// TIA Portal V20 export
ORGANIZATION_BLOCK "Main"   // OB124, LAD, ProgramCycle
TITLE = "Main Program Sweep (Cycle)"
// stored: Namespace PFE, SetENOAutomatically false
   VAR_INPUT
      Initial_Call : Bool;   // Initial call of this OB
      Remanence : Bool;   // =True, if remanent data are available
   END_VAR
   VAR_TEMP
      tempEnable : Bool;   // Replace with the user tags
      tempFilter : Bool;   // Replace with the user tags
      tempValid : Bool;   // Replace with the user tags
      tempBusy : Bool;   // Replace with the user tags
      tempError : Bool;   // Replace with the user tags
      tempStatus : Word;   // Replace with the user tags
   END_VAR
BEGIN

REGION Network 1: Calling Digital Event Handler
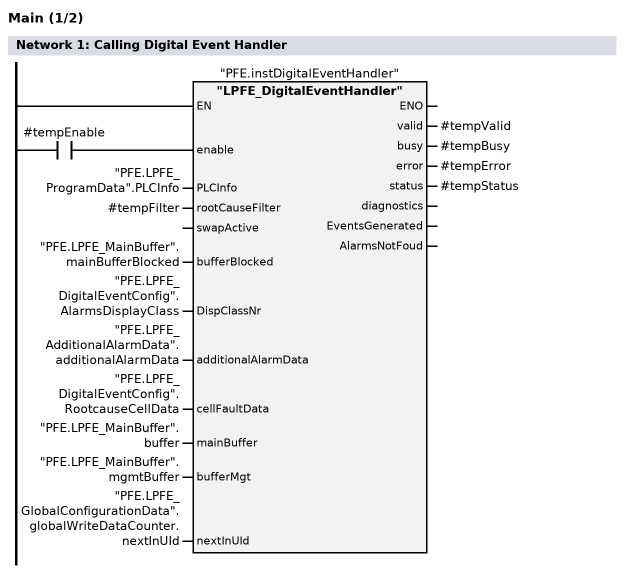
   RUNG wire#powerrail
      "PFE.instDigitalEventHandler"(enable := wire#w1, PLCInfo := "PFE.LPFE_ProgramData".PLCInfo, rootCauseFilter := #tempFilter, swapActive :=, bufferBlocked := "PFE.LPFE_MainBuffer".mainBufferBlocked, DispClassNr := "PFE.LPFE_DigitalEventConfig".AlarmsDisplayClass, additionalAlarmData := "PFE.LPFE_AdditionalAlarmData".additionalAlarmData, cellFaultData := "PFE.LPFE_DigitalEventConfig".RootcauseCellData, mainBuffer := "PFE.LPFE_MainBuffer".buffer, bufferMgt := "PFE.LPFE_MainBuffer".mgmtBuffer, nextInUId := "PFE.LPFE_GlobalConfigurationData".globalWriteDataCounter.nextInUId, valid => #tempValid, busy => #tempBusy, error => #tempError, status => #tempStatus, diagnostics =>, EventsGenerated =>, AlarmsNotFoud =>)
   END_RUNG
   RUNG wire#powerrail
      Contact( #tempEnable )
   END_RUNG wire#w1
   // the same network as SCL:
   "PFE.instDigitalEventHandler"(enable := #tempEnable,   // "LPFE_DigitalEventHandler"
                           PLCInfo := "PFE.LPFE_ProgramData".PLCInfo,
                           rootCauseFilter := #tempFilter,
                           bufferBlocked := "PFE.LPFE_MainBuffer".mainBufferBlocked,
                           DispClassNr := "PFE.LPFE_DigitalEventConfig".AlarmsDisplayClass,
                           additionalAlarmData := "PFE.LPFE_AdditionalAlarmData".additionalAlarmData,
                           cellFaultData := "PFE.LPFE_DigitalEventConfig".RootcauseCellData,
                           mainBuffer := "PFE.LPFE_MainBuffer".buffer,
                           bufferMgt := "PFE.LPFE_MainBuffer".mgmtBuffer,
                           nextInUId := "PFE.LPFE_GlobalConfigurationData".globalWriteDataCounter.nextInUId,
                           valid => #tempValid,
                           busy => #tempBusy,
                           error => #tempError,
                           status => #tempStatus);
END_REGION

REGION Network 2: Calling PFE Backbone Strucuture
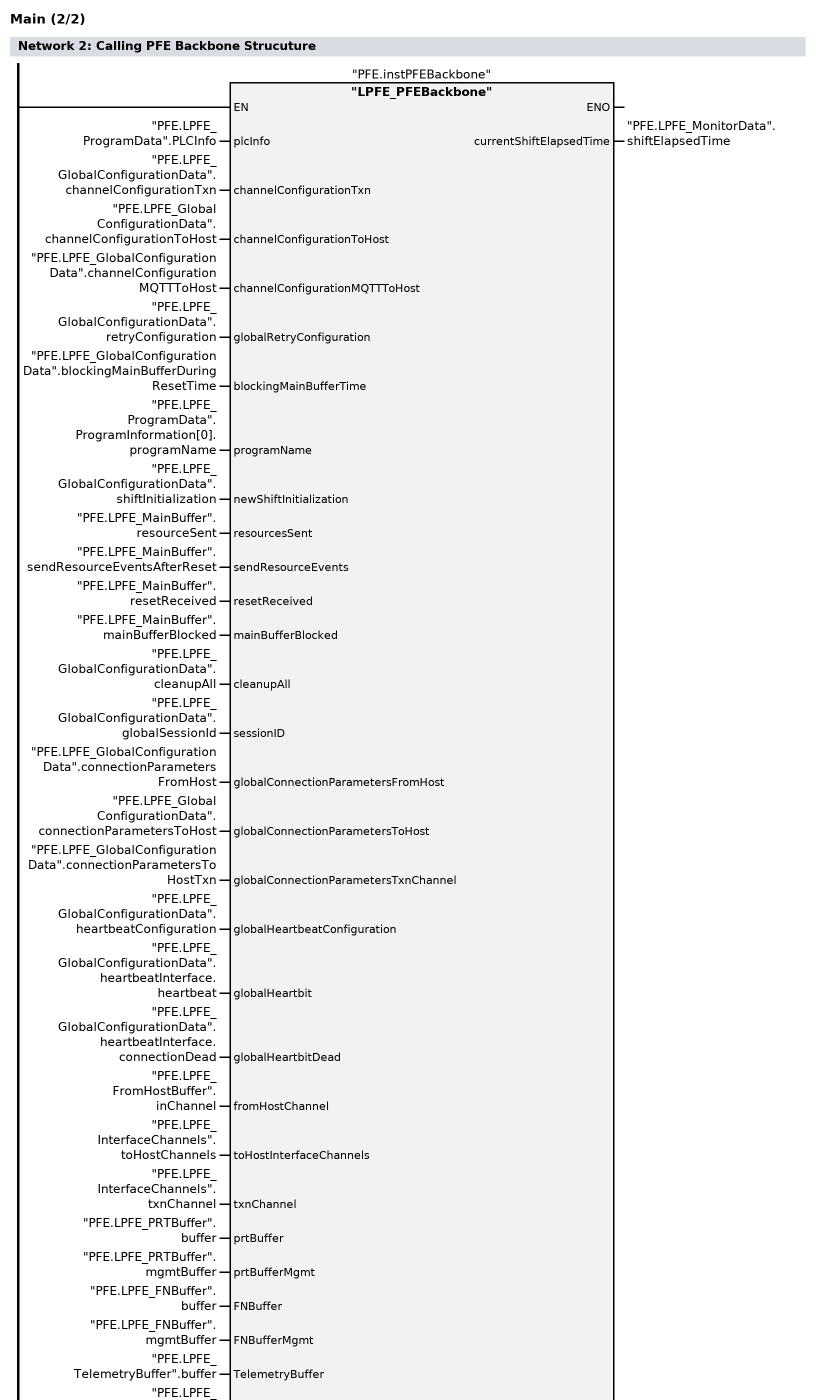
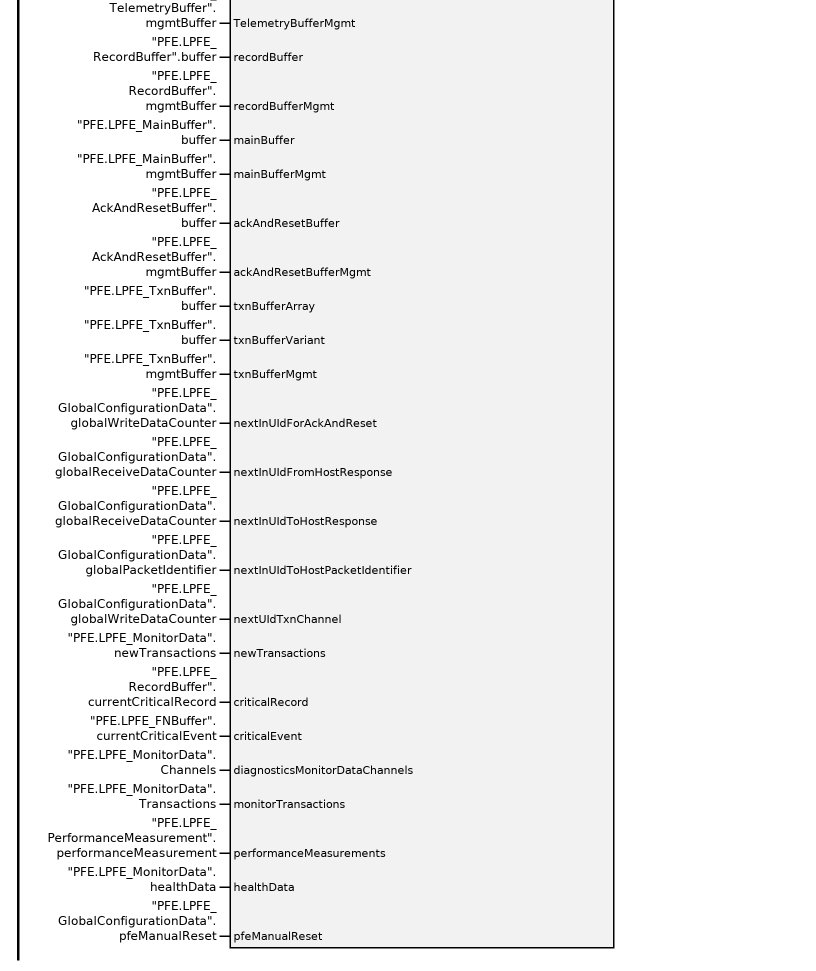
   RUNG wire#powerrail
      "PFE.instPFEBackbone"(plcInfo := "PFE.LPFE_ProgramData".PLCInfo, channelConfigurationTxn := "PFE.LPFE_GlobalConfigurationData".channelConfigurationTxn, channelConfigurationToHost := "PFE.LPFE_GlobalConfigurationData".channelConfigurationToHost, channelConfigurationMQTTToHost := "PFE.LPFE_GlobalConfigurationData".channelConfigurationMQTTToHost, globalRetryConfiguration := "PFE.LPFE_GlobalConfigurationData".retryConfiguration, blockingMainBufferTime := "PFE.LPFE_GlobalConfigurationData".blockingMainBufferDuringResetTime, programName := "PFE.LPFE_ProgramData".ProgramInformation[0].programName, newShiftInitialization := "PFE.LPFE_GlobalConfigurationData".shiftInitialization, resourcesSent := "PFE.LPFE_MainBuffer".resourceSent, sendResourceEvents := "PFE.LPFE_MainBuffer".sendResourceEventsAfterReset, resetReceived := "PFE.LPFE_MainBuffer".resetReceived, mainBufferBlocked := "PFE.LPFE_MainBuffer".mainBufferBlocked, cleanupAll := "PFE.LPFE_GlobalConfigurationData".cleanupAll, sessionID := "PFE.LPFE_GlobalConfigurationData".globalSessionId, globalConnectionParametersFromHost := "PFE.LPFE_GlobalConfigurationData".connectionParametersFromHost, globalConnectionParametersToHost := "PFE.LPFE_GlobalConfigurationData".connectionParametersToHost, globalConnectionParametersTxnChannel := "PFE.LPFE_GlobalConfigurationData".connectionParametersToHostTxn, globalHeartbeatConfiguration := "PFE.LPFE_GlobalConfigurationData".heartbeatConfiguration, globalHeartbit := "PFE.LPFE_GlobalConfigurationData".heartbeatInterface.heartbeat, globalHeartbitDead := "PFE.LPFE_GlobalConfigurationData".heartbeatInterface.connectionDead, fromHostChannel := "PFE.LPFE_FromHostBuffer".inChannel, toHostInterfaceChannels := "PFE.LPFE_InterfaceChannels".toHostChannels, txnChannel := "PFE.LPFE_InterfaceChannels".txnChannel, prtBuffer := "PFE.LPFE_PRTBuffer".buffer, prtBufferMgmt := "PFE.LPFE_PRTBuffer".mgmtBuffer, FNBuffer := "PFE.LPFE_FNBuffer".buffer, FNBufferMgmt := "PFE.LPFE_FNBuffer".mgmtBuffer, TelemetryBuffer := "PFE.LPFE_TelemetryBuffer".buffer, TelemetryBufferMgmt := "PFE.LPFE_TelemetryBuffer".mgmtBuffer, recordBuffer := "PFE.LPFE_RecordBuffer".buffer, recordBufferMgmt := "PFE.LPFE_RecordBuffer".mgmtBuffer, mainBuffer := "PFE.LPFE_MainBuffer".buffer, mainBufferMgmt := "PFE.LPFE_MainBuffer".mgmtBuffer, ackAndResetBuffer := "PFE.LPFE_AckAndResetBuffer".buffer, ackAndResetBufferMgmt := "PFE.LPFE_AckAndResetBuffer".mgmtBuffer, txnBufferArray := "PFE.LPFE_TxnBuffer".buffer, txnBufferVariant := "PFE.LPFE_TxnBuffer".buffer, txnBufferMgmt := "PFE.LPFE_TxnBuffer".mgmtBuffer, nextInUIdForAckAndReset := "PFE.LPFE_GlobalConfigurationData".globalWriteDataCounter, nextInUIdFromHostResponse := "PFE.LPFE_GlobalConfigurationData".globalReceiveDataCounter, nextInUIdToHostResponse := "PFE.LPFE_GlobalConfigurationData".globalReceiveDataCounter, nextInUIdToHostPacketIdentifier := "PFE.LPFE_GlobalConfigurationData".globalPacketIdentifier, nextUIdTxnChannel := "PFE.LPFE_GlobalConfigurationData".globalWriteDataCounter, newTransactions := "PFE.LPFE_MonitorData".newTransactions, criticalRecord := "PFE.LPFE_RecordBuffer".currentCriticalRecord, criticalEvent := "PFE.LPFE_FNBuffer".currentCriticalEvent, diagnosticsMonitorDataChannels := "PFE.LPFE_MonitorData".Channels, monitorTransactions := "PFE.LPFE_MonitorData".Transactions, performanceMeasurements := "PFE.LPFE_PerformanceMeasurement".performanceMeasurement, healthData := "PFE.LPFE_MonitorData".healthData, pfeManualReset := "PFE.LPFE_GlobalConfigurationData".pfeManualReset, currentShiftElapsedTime => "PFE.LPFE_MonitorData".shiftElapsedTime)
   END_RUNG
   // the same network as SCL:
   "PFE.instPFEBackbone"(plcInfo := "PFE.LPFE_ProgramData".PLCInfo,   // "LPFE_PFEBackbone"
                         channelConfigurationTxn := "PFE.LPFE_GlobalConfigurationData".channelConfigurationTxn,
                         channelConfigurationToHost := "PFE.LPFE_GlobalConfigurationData".channelConfigurationToHost,
                         channelConfigurationMQTTToHost := "PFE.LPFE_GlobalConfigurationData".channelConfigurationMQTTToHost,
                         globalRetryConfiguration := "PFE.LPFE_GlobalConfigurationData".retryConfiguration,
                         blockingMainBufferTime := "PFE.LPFE_GlobalConfigurationData".blockingMainBufferDuringResetTime,
                         programName := "PFE.LPFE_ProgramData".ProgramInformation[0].programName,
                         newShiftInitialization := "PFE.LPFE_GlobalConfigurationData".shiftInitialization,
                         resourcesSent := "PFE.LPFE_MainBuffer".resourceSent,
                         sendResourceEvents := "PFE.LPFE_MainBuffer".sendResourceEventsAfterReset,
                         resetReceived := "PFE.LPFE_MainBuffer".resetReceived,
                         mainBufferBlocked := "PFE.LPFE_MainBuffer".mainBufferBlocked,
                         cleanupAll := "PFE.LPFE_GlobalConfigurationData".cleanupAll,
                         sessionID := "PFE.LPFE_GlobalConfigurationData".globalSessionId,
                         globalConnectionParametersFromHost := "PFE.LPFE_GlobalConfigurationData".connectionParametersFromHost,
                         globalConnectionParametersToHost := "PFE.LPFE_GlobalConfigurationData".connectionParametersToHost,
                         globalConnectionParametersTxnChannel := "PFE.LPFE_GlobalConfigurationData".connectionParametersToHostTxn,
                         globalHeartbeatConfiguration := "PFE.LPFE_GlobalConfigurationData".heartbeatConfiguration,
                         globalHeartbit := "PFE.LPFE_GlobalConfigurationData".heartbeatInterface.heartbeat,
                         globalHeartbitDead := "PFE.LPFE_GlobalConfigurationData".heartbeatInterface.connectionDead,
                         fromHostChannel := "PFE.LPFE_FromHostBuffer".inChannel,
                         toHostInterfaceChannels := "PFE.LPFE_InterfaceChannels".toHostChannels,
                         txnChannel := "PFE.LPFE_InterfaceChannels".txnChannel,
                         prtBuffer := "PFE.LPFE_PRTBuffer".buffer,
                         prtBufferMgmt := "PFE.LPFE_PRTBuffer".mgmtBuffer,
                         FNBuffer := "PFE.LPFE_FNBuffer".buffer,
                         FNBufferMgmt := "PFE.LPFE_FNBuffer".mgmtBuffer,
                         TelemetryBuffer := "PFE.LPFE_TelemetryBuffer".buffer,
                         TelemetryBufferMgmt := "PFE.LPFE_TelemetryBuffer".mgmtBuffer,
                         recordBuffer := "PFE.LPFE_RecordBuffer".buffer,
                         recordBufferMgmt := "PFE.LPFE_RecordBuffer".mgmtBuffer,
                         mainBuffer := "PFE.LPFE_MainBuffer".buffer,
                         mainBufferMgmt := "PFE.LPFE_MainBuffer".mgmtBuffer,
                         ackAndResetBuffer := "PFE.LPFE_AckAndResetBuffer".buffer,
                         ackAndResetBufferMgmt := "PFE.LPFE_AckAndResetBuffer".mgmtBuffer,
                         txnBufferArray := "PFE.LPFE_TxnBuffer".buffer,
                         txnBufferVariant := "PFE.LPFE_TxnBuffer".buffer,
                         txnBufferMgmt := "PFE.LPFE_TxnBuffer".mgmtBuffer,
                         nextInUIdForAckAndReset := "PFE.LPFE_GlobalConfigurationData".globalWriteDataCounter,
                         nextInUIdFromHostResponse := "PFE.LPFE_GlobalConfigurationData".globalReceiveDataCounter,
                         nextInUIdToHostResponse := "PFE.LPFE_GlobalConfigurationData".globalReceiveDataCounter,
                         nextInUIdToHostPacketIdentifier := "PFE.LPFE_GlobalConfigurationData".globalPacketIdentifier,
                         nextUIdTxnChannel := "PFE.LPFE_GlobalConfigurationData".globalWriteDataCounter,
                         newTransactions := "PFE.LPFE_MonitorData".newTransactions,
                         criticalRecord := "PFE.LPFE_RecordBuffer".currentCriticalRecord,
                         criticalEvent := "PFE.LPFE_FNBuffer".currentCriticalEvent,
                         diagnosticsMonitorDataChannels := "PFE.LPFE_MonitorData".Channels,
                         monitorTransactions := "PFE.LPFE_MonitorData".Transactions,
                         performanceMeasurements := "PFE.LPFE_PerformanceMeasurement".performanceMeasurement,
                         healthData := "PFE.LPFE_MonitorData".healthData,
                         pfeManualReset := "PFE.LPFE_GlobalConfigurationData".pfeManualReset,
                         currentShiftElapsedTime => "PFE.LPFE_MonitorData".shiftElapsedTime);
END_REGION
END_ORGANIZATION_BLOCK
